# EPICS autosave request: dxp/tags/R1-3beta2/iocBoot/iocDxpLinux_RC/auto_settings_med.req
file "simple_mca_settings.req",                P=dxpLinux:med:, M=mca1
file "dxp_settings.req",                P=dxpLinux:med:, R=dxp1
